# EPICS substitutions: pvNotepadApp/Db/ao_10.substitutions
#Substitutions for 10 records
file ao.template
{
    pattern { RECORD             }
            { $(HUTCH):NOTE:DOUBLE:01 }
            { $(HUTCH):NOTE:DOUBLE:02 }
            { $(HUTCH):NOTE:DOUBLE:03 }
            { $(HUTCH):NOTE:DOUBLE:04 }
            { $(HUTCH):NOTE:DOUBLE:05 }
            { $(HUTCH):NOTE:DOUBLE:06 }
            { $(HUTCH):NOTE:DOUBLE:07 }
            { $(HUTCH):NOTE:DOUBLE:08 }
            { $(HUTCH):NOTE:DOUBLE:09 }
            { $(HUTCH):NOTE:DOUBLE:10 }
}
